TYPE "EFC_STATUS_WORD"
VERSION : 0.1
// Block: EFC_STATUS_WORD
   STRUCT
      ErrorCode0 : Bool;
      ErrorCode1 : Bool;
      ErrorCode2 : Bool;
      ErrorCode3 : Bool;
      ErrorCode4 : Bool;
      ErrorCode5 : Bool;
      ErrorCode6 : Bool;
      ErrorCode7 : Bool;
      Reverse : Bool;
      Running : Bool;
      Jogging : Bool;
      Accelerating : Bool;
      Decelerating : Bool;
      OverVoltage : Bool;
      OverCurrent : Bool;
      Error : Bool;
   END_STRUCT;

END_TYPE
